PROGRAM P_Control
VAR
	fbStarter: FB_StartingAlarm;
	FB_Debounce_0: FB_Debounce;
	fbDebounce: FB_Debounce;
	fbContactor: FB_Contactor;
	simContactor: FB_Debounce;
END_VAR

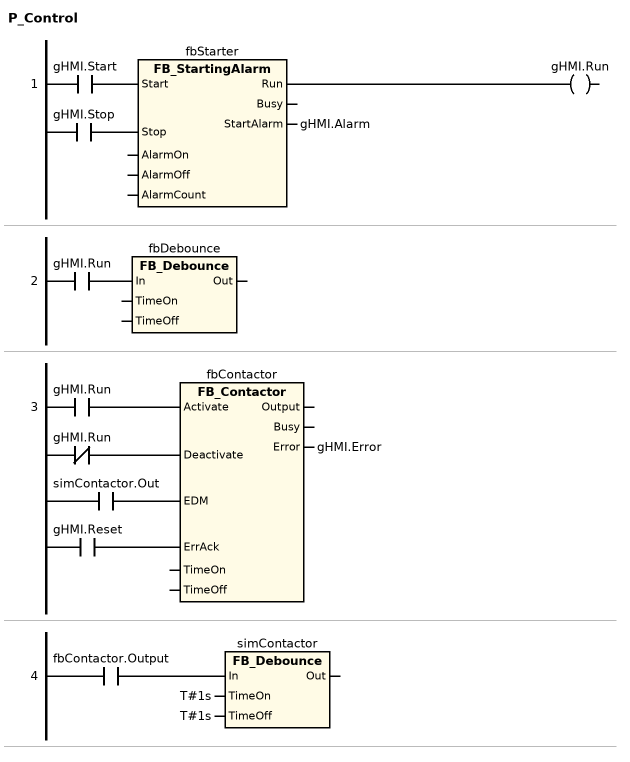
// NETWORK 1
fbStarter(Start := gHMI.Start, Stop := gHMI.Stop, StartAlarm => gHMI.Alarm); // FB_StartingAlarm
gHMI.Run := fbStarter.Run;

// NETWORK 2
fbDebounce(In := gHMI.Run); // FB_Debounce

// NETWORK 3
fbContactor(
    Activate := gHMI.Run,
    Deactivate := NOT gHMI.Run,
    EDM := simContactor.Out,
    ErrAck := gHMI.Reset,
    Error => gHMI.Error); // FB_Contactor

// NETWORK 4
simContactor(In := fbContactor.Output, TimeOn := T#1s, TimeOff := T#1s); // FB_Debounce

END_PROGRAM

(* stored: Version 1.1.0.1, ProductVersion 3.1.4024.12
   POU P_Control: Id {d7d0d404-2b8f-4922-b3b9-8421354cbc9f}, SpecialFunc None *)
